FUNCTION_BLOCK FB_SetTargetValues
VAR_INPUT
END_VAR
VAR_OUTPUT
END_VAR
VAR
	nCallCount : UINT;
	nTargetValues : ARRAY[0..2] OF ST_TargetValueDataType;
END_VAR

{attribute 'TcRpcEnable' := '1'}
METHOD Abort : HRESULT
VAR_INPUT
END_VAR
END_METHOD

PROPERTY bBusy : BOOL
GET
END_GET
SET
END_SET
END_PROPERTY

{attribute 'TcRpcEnable' := '1'}
METHOD CheckState : HRESULT
VAR_INPUT
	hdl : UDINT;
END_VAR
END_METHOD

PROPERTY hrError : HRESULT
GET
END_GET
SET
END_SET
END_PROPERTY

{attribute 'TcRpcEnable' := '1'}
METHOD Start : HRESULT
VAR_INPUT
	TargetValues : ARRAY[0..2] OF ST_TargetValueDataType;
END_VAR
nCallCount := nCallCount + 1;
nTargetValues[0] := TargetValues[0];
nTargetValues[1] := TargetValues[1];
nTargetValues[2] := TargetValues[2];
END_METHOD

END_FUNCTION_BLOCK

(* stored: Version 1.1.0.1, ProductVersion 3.1.4024.3
   POU FB_SetTargetValues: Id {c651fa1d-c78e-4f2b-b3f3-7b277b8ff218}, SpecialFunc None
   Method Abort: Id {b8a4f22f-739b-4bf6-accd-82557357612c}
   Property bBusy: Id {48827013-2ae1-47b8-97b0-d0a2d3d9bd57}
   Get Get: Id {e891cf25-af0a-4e30-bb15-4751ed3f51e6}
   Set Set: Id {5b39db1d-fa88-4a9c-80f5-bf138e35f613}
   Method CheckState: Id {a3b66854-84bf-427a-8a9f-f808be302837}
   Property hrError: Id {f6925bb3-818e-4e2f-9b51-2c74e72dfa2f}
   Get Get: Id {039c9d98-07b2-4c8f-8391-5f9965bb199c}
   Set Set: Id {89856b64-6315-48d1-ac41-ecccbed78517}
   Method Start: Id {4c922c5b-a284-49cb-9736-936debe52028} *)
